{attribute 'GeneratedUsingTerminal: EP9128-0021-0017'}
{attribute addProperty BoxType "EP9128-0021-0017"}
{attribute addProperty Id "A_0010_EP9128_0021_0018A_0010_EP9128_0021_0018_AD796AAA583A_0007_EP9128_0021_0017_2_EP9128_1021EP9128_AB5A94672A_0007_EP9128_0021_0017_3_EP9128_2021EP9128_AB5A94672"}
{attribute addProperty CRC "3669521390"}
{attribute addProperty Size "587"}
TYPE A_0007_EP9128_0021_0017_DAB873EE EXTENDS EP9128_AB5A9467 :
STRUCT
	{attribute addProperty Name "A_0010_EP9128_0021_0018"}
	{attribute addProperty PreviousPort "A_0007(EP9128-0021-0017) : D"}
	A_0010_EP9128_0021_0018 : A_0010_EP9128_0021_0018_AD796AAA;
	{attribute addProperty Name "A_0007_EP9128_0021_0017_2_EP9128_1021"}
	{attribute addProperty PreviousPort "A_0007(EP9128-0021-0017) : C"}
	A_0007_EP9128_0021_0017_2_EP9128_1021 : EP9128_AB5A9467;
	{attribute addProperty Name "A_0007_EP9128_0021_0017_3_EP9128_2021"}
	{attribute addProperty PreviousPort "A_0007(EP9128-0021-0017)_2 (EP9128-1021) : C"}
	A_0007_EP9128_0021_0017_3_EP9128_2021 : EP9128_AB5A9467;
END_STRUCT
END_TYPE

(* stored: Version 1.2.0.0, ProductVersion 3.1.4024.9
   DUT A_0007_EP9128_0021_0017_DAB873EE: Id {c112611b-90f8-4ea4-814c-51efcc71f156} *)
